FUNCTION_BLOCK FB_Blokgolf
VAR_INPUT
END_VAR
VAR_OUTPUT
END_VAR
VAR
	_timer1 : TP;
	_timer2 : TP;
	bEnabled: BOOL;
END_VAR

_timer1.IN := bEnabled AND NOT _timer2.Q;
_timer1();

_timer2.IN := bEnabled AND NOT _timer1.Q;
_timer2();

PROPERTY PUBLIC bSignalOut : BOOL
GET
END_GET
SET
END_SET
END_PROPERTY

METHOD PUBLIC M_Start
VAR_INPUT
	onTime : TIME;
	offTime : TIME;
END_VAR
bEnabled := TRUE;
_timer1.PT := onTime;
_timer2.PT := offTime;
END_METHOD

METHOD PUBLIC M_Stop
VAR_INPUT
END_VAR
bEnabled := false;
END_METHOD

PROPERTY PUBLIC nCounter : REAL
GET
END_GET
SET
END_SET
END_PROPERTY

END_FUNCTION_BLOCK

(* stored: Version 1.1.0.1, ProductVersion 3.1.4024.13
   POU FB_Blokgolf: Id {d0b27e9a-7cde-4b2e-a891-902789c8648a}, SpecialFunc None
   Property bSignalOut: Id {28d69959-e79d-41a9-8ffe-7579100c444f}
   Get Get: Id {291c1f72-9207-4cec-8a34-6059f1bff2c1}
   Set Set: Id {4926ffb8-daf8-4c4f-938e-dfb7ea85ee92}
   Method M_Start: Id {d7473e49-bd23-4ff1-8062-541eb712e25e}
   Method M_Stop: Id {189d4a1f-c273-4665-af82-f2d525d6f123}
   Property nCounter: Id {1757287f-c614-468e-986e-353590e49607}
   Get Get: Id {479e1dee-2000-4d97-b0a5-faa09234d9cf}
   Set Set: Id {02650336-76ed-4272-a435-cbae06038377} *)
